// SIMATIC STEP 7 (V5.x) project S7_Demo
// CPU: CPU 313C-2 DP
// station: P_ADR_BUS
// station: Hardware
// station: SIMATIC 300 Station
// program: S7 Program(2)

SYMBOL_TABLE
"I0.0"	I 0.0	BOOL	// start
"I0.1"	I 0.1	BOOL	// stop
"I1.1"	I 1.1	BOOL	// CB HOP TREN BANG TRUYEN
"I1.2"	I 1.2	BOOL	// CB DEM SP
"I1.3"	I 1.3	BOOL	// CB VT HOP
"I7.0"	I 7.0	BOOL	// reset
"M0.0"	M 0.0	BOOL	// ON
"M0.1"	M 0.1	BOOL	// T/H HOP DEN  VT 2P
"M0.2"	M 0.2	BOOL	// STOP
"M0.3"	M 0.3	BOOL	// BANG CHUYEN SP
"M0.4"	M 0.4	BOOL	// DU SO HOP
"M0.5"	M 0.5	BOOL	// BIT NHO DA DEM 2P
"M1.1"	M 1.1	BOOL	// KICH TIMER 2
"M1.3"	M 1.3	BOOL	// DU SO LUONG SP/HOP
"M2.1"	M 2.1	BOOL	// COI VA DEN BAO LOI
"Q1.1"	Q 1.1	BOOL	// Bang truyen hop
"Q1.2"	Q 1.2	BOOL	// Bang chuyen sp
"Q2.0"	Q 2.0	BOOL	// COI VA DEN BAO LOI
END_SYMBOL_TABLE

ORGANIZATION_BLOCK OB 1
TITLE = NHOM9
//BO DIEU KHIEN HE THONG DONG GOI SAN PHAM
VERSION : 0.1
VAR_TEMP
  OB1_EV_CLASS : BYTE ;	//Bits 0-3 = 1 (Coming event), Bits 4-7 = 1 (Event class 1)
  OB1_SCAN_1 : BYTE ;	//1 (Cold restart scan 1 of OB 1), 3 (Scan 2-n of OB 1)
  OB1_PRIORITY : BYTE ;	//Priority of OB Execution
  OB1_OB_NUMBR : BYTE ;	//1 (Organization block 1, OB1)
  OB1_RESERVED_1 : BYTE ;	//Reserved for system
  OB1_RESERVED_2 : BYTE ;	//Reserved for system
  OB1_PREV_CYCLE : INT ;	//Cycle time of previous OB1 scan (milliseconds)
  OB1_MIN_CYCLE : INT ;	//Minimum cycle time of OB1 (milliseconds)
  OB1_MAX_CYCLE : INT ;	//Maximum cycle time of OB1 (milliseconds)
  OB1_DATE_TIME : DATE_AND_TIME ;	//Date and time OB1 started
END_VAR
BEGIN
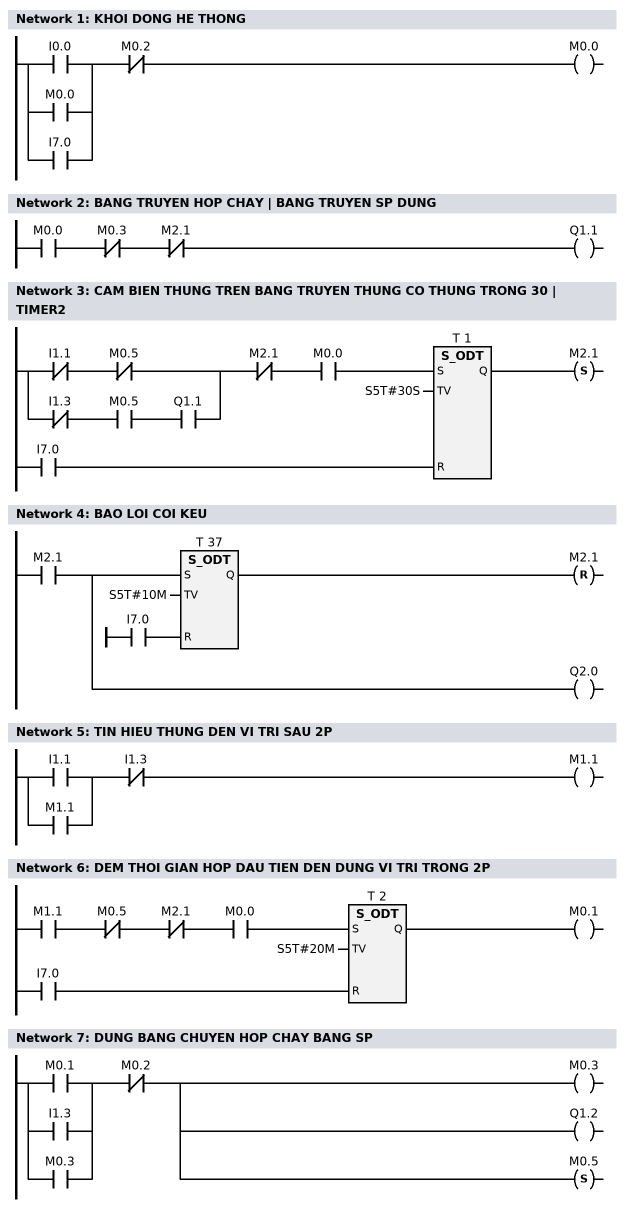
NETWORK
TITLE = KHOI DONG HE THONG
      A(;
      O     "I0.0";
      O     "M0.0";
      O     "I7.0";
      );
      AN    "M0.2";
      =     "M0.0";
NETWORK
TITLE = BANG TRUYEN HOP CHAY | BANG TRUYEN SP DUNG 
      A     "M0.0";
      AN    "M0.3";
      AN    "M2.1";
      =     "Q1.1";
NETWORK
TITLE = CAM BIEN THUNG TREN BANG TRUYEN THUNG CO THUNG TRONG 30 | TIMER2
      A(;
      AN    "I1.1";
      AN    "M0.5";
      O;
      AN    "I1.3";
      A     "M0.5";
      A     "Q1.1";
      );
      AN    "M2.1";
      A     "M0.0";
      L     S5T#30S;
      SD    T 1;
      A     "I7.0";
      R     T 1;
      NOP   0;
      NOP   0;
      A     T 1;
      S     "M2.1";
NETWORK
TITLE = BAO LOI COI KEU
      A     "M2.1";
      =     L 20.0;
      A     L 20.0;
      L     S5T#10M;
      SD    T 37;
      A     "I7.0";
      R     T 37;
      NOP   0;
      NOP   0;
      A     T 37;
      R     "M2.1";
      A     L 20.0;
      BLD   102;
      =     "Q2.0";
NETWORK
TITLE = TIN HIEU THUNG DEN VI TRI SAU 2P
      A(;
      O     "I1.1";
      O     "M1.1";
      );
      AN    "I1.3";
      =     "M1.1";
NETWORK
TITLE = DEM THOI GIAN HOP DAU TIEN DEN DUNG VI TRI TRONG 2P
      A     "M1.1";
      AN    "M0.5";
      AN    "M2.1";
      A     "M0.0";
      L     S5T#20M;
      SD    T 2;
      A     "I7.0";
      R     T 2;
      NOP   0;
      NOP   0;
      A     T 2;
      =     "M0.1";
NETWORK
TITLE = DUNG BANG CHUYEN HOP CHAY BANG SP
      A(;
      O     "M0.1";
      O     "I1.3";
      O     "M0.3";
      );
      AN    "M0.2";
      =     "M0.3";
      =     "Q1.2";
      S     "M0.5";
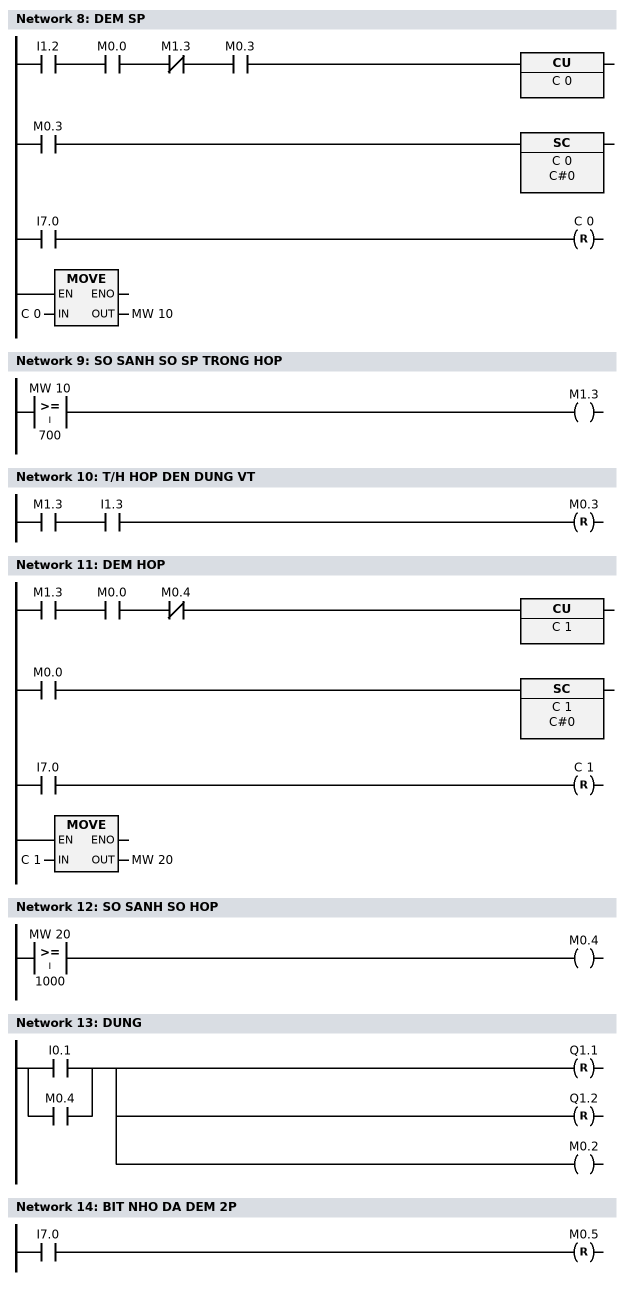
NETWORK
TITLE = DEM SP
      A     "I1.2";
      A     "M0.0";
      AN    "M1.3";
      A     "M0.3";
      CU    C 0;
      BLD   101;
      A     "M0.3";
      L     C#0;
      S     C 0;
      A     "I7.0";
      R     C 0;
      L     C 0;
      T     MW 10;
      NOP   0;
      NOP   0;
NETWORK
TITLE = SO SANH SO SP TRONG HOP 
      L     MW 10;
      L     700;
      >=I;
      =     "M1.3";
NETWORK
TITLE = T/H HOP DEN DUNG VT
      A     "M1.3";
      A     "I1.3";
      R     "M0.3";
NETWORK
TITLE = DEM HOP
      A     "M1.3";
      A     "M0.0";
      AN    "M0.4";
      CU    C 1;
      BLD   101;
      A     "M0.0";
      L     C#0;
      S     C 1;
      A     "I7.0";
      R     C 1;
      L     C 1;
      T     MW 20;
      NOP   0;
      NOP   0;
NETWORK
TITLE = SO SANH SO HOP
      L     MW 20;
      L     1000;
      >=I;
      =     "M0.4";
NETWORK
TITLE = DUNG
      O     "I0.1";
      O     "M0.4";
      R     "Q1.1";
      R     "Q1.2";
      =     "M0.2";
NETWORK
TITLE = BIT NHO DA DEM 2P
      A     "I7.0";
      R     "M0.5";
END_ORGANIZATION_BLOCK
